//Alarm Word 24
(* uncomment when instrument is ready
Alarms_DB.AlarmWord_24.AlarmWord.0 := Trips_DB.Coil[9].ChargeRelay_FailtoClose; 
Alarms_DB.AlarmWord_24.AlarmWord.1 := Trips_DB.Coil[9].ChargeRelay_FailtoOpen;
Alarms_DB.AlarmWord_24.AlarmWord.2 := Trips_DB.Coil[10].ChargeRelay_FailtoClose;
Alarms_DB.AlarmWord_24.AlarmWord.3 := Trips_DB.Coil[10].ChargeRelay_FailtoOpen;
Alarms_DB.AlarmWord_24.AlarmWord.4 := Trips_DB.Coil[1].ACInterlockRelayFailedtoClose;
Alarms_DB.AlarmWord_24.AlarmWord.5 := Trips_DB.Coil[1].ACInterlockRelayFailedtoOpen;
Alarms_DB.AlarmWord_24.AlarmWord.6 := Trips_DB.Coil[2].ACInterlockRelayFailedtoClose;
Alarms_DB.AlarmWord_24.AlarmWord.7 := Trips_DB.Coil[2].ACInterlockRelayFailedtoOpen;
Alarms_DB.AlarmWord_24.AlarmWord.8 := Trips_DB.Coil[3].ACInterlockRelayFailedtoClose;
Alarms_DB.AlarmWord_24.AlarmWord.9 := Trips_DB.Coil[3].ACInterlockRelayFailedtoOpen;
Alarms_DB.AlarmWord_24.AlarmWord.10 := Trips_DB.Coil[4].ACInterlockRelayFailedtoClose;
Alarms_DB.AlarmWord_24.AlarmWord.11 := Trips_DB.Coil[4].ACInterlockRelayFailedtoOpen;
Alarms_DB.AlarmWord_24.AlarmWord.12 := Trips_DB.Coil[5].ACInterlockRelayFailedtoClose;
Alarms_DB.AlarmWord_24.AlarmWord.13 := Trips_DB.Coil[5].ACInterlockRelayFailedtoOpen;
Alarms_DB.AlarmWord_24.AlarmWord.14 := Trips_DB.Coil[6].ACInterlockRelayFailedtoClose;
Alarms_DB.AlarmWord_24.AlarmWord.15 := Trips_DB.Coil[6].ACInterlockRelayFailedtoOpen;
*)
//Alarm Word 24 msg
alarms[368](evtEntry:= Tc_Events.AlarmWord24.b0, bEvt:= Alarms_DB.AlarmWord_24.AlarmWord.0, bConfirm:= bConfirm);
alarms[369](evtEntry:= Tc_Events.AlarmWord24.b1, bEvt:= Alarms_DB.AlarmWord_24.AlarmWord.1, bConfirm:= bConfirm);
alarms[370](evtEntry:= Tc_Events.AlarmWord24.b2, bEvt:= Alarms_DB.AlarmWord_24.AlarmWord.2, bConfirm:= bConfirm);
alarms[371](evtEntry:= Tc_Events.AlarmWord24.b3, bEvt:= Alarms_DB.AlarmWord_24.AlarmWord.3, bConfirm:= bConfirm);
alarms[372](evtEntry:= Tc_Events.AlarmWord24.b4, bEvt:= Alarms_DB.AlarmWord_24.AlarmWord.4, bConfirm:= bConfirm);
alarms[373](evtEntry:= Tc_Events.AlarmWord24.b5, bEvt:= Alarms_DB.AlarmWord_24.AlarmWord.5, bConfirm:= bConfirm);
alarms[374](evtEntry:= Tc_Events.AlarmWord24.b6, bEvt:= Alarms_DB.AlarmWord_24.AlarmWord.6, bConfirm:= bConfirm);
alarms[375](evtEntry:= Tc_Events.AlarmWord24.b7, bEvt:= Alarms_DB.AlarmWord_24.AlarmWord.7, bConfirm:= bConfirm);
alarms[376](evtEntry:= Tc_Events.AlarmWord24.b8, bEvt:= Alarms_DB.AlarmWord_24.AlarmWord.8, bConfirm:= bConfirm);
alarms[377](evtEntry:= Tc_Events.AlarmWord24.b9, bEvt:= Alarms_DB.AlarmWord_24.AlarmWord.9, bConfirm:= bConfirm);
alarms[378](evtEntry:= Tc_Events.AlarmWord24.b10, bEvt:= Alarms_DB.AlarmWord_24.AlarmWord.10, bConfirm:= bConfirm);
alarms[379](evtEntry:= Tc_Events.AlarmWord24.b11, bEvt:= Alarms_DB.AlarmWord_24.AlarmWord.11, bConfirm:= bConfirm);
alarms[380](evtEntry:= Tc_Events.AlarmWord24.b12, bEvt:= Alarms_DB.AlarmWord_24.AlarmWord.12, bConfirm:= bConfirm);
alarms[381](evtEntry:= Tc_Events.AlarmWord24.b13, bEvt:= Alarms_DB.AlarmWord_24.AlarmWord.13, bConfirm:= bConfirm);
alarms[382](evtEntry:= Tc_Events.AlarmWord24.b14, bEvt:= Alarms_DB.AlarmWord_24.AlarmWord.14, bConfirm:= bConfirm);
alarms[383](evtEntry:= Tc_Events.AlarmWord24.b15, bEvt:= Alarms_DB.AlarmWord_24.AlarmWord.15, bConfirm:= bConfirm);

//Alarm Word 25
(* uncomment when instrument is ready
Alarms_DB.AlarmWord_25.AlarmWord.0 := Trips_DB.Coil[7].ACInterlockRelayFailedtoClose;
Alarms_DB.AlarmWord_25.AlarmWord.1 := Trips_DB.Coil[7].ACInterlockRelayFailedtoOpen;
Alarms_DB.AlarmWord_25.AlarmWord.2 := Trips_DB.Coil[8].ACInterlockRelayFailedtoClose;
Alarms_DB.AlarmWord_25.AlarmWord.3 := Trips_DB.Coil[8].ACInterlockRelayFailedtoOpen;
Alarms_DB.AlarmWord_25.AlarmWord.4 := Trips_DB.Coil[9].ACInterlockRelayFailedtoClose;
Alarms_DB.AlarmWord_25.AlarmWord.5 := Trips_DB.Coil[9].ACInterlockRelayFailedtoOpen;
Alarms_DB.AlarmWord_25.AlarmWord.6 := Trips_DB.Coil[10].ACInterlockRelayFailedtoClose;
Alarms_DB.AlarmWord_25.AlarmWord.7 := Trips_DB.Coil[10].ACInterlockRelayFailedtoOpen;
Alarms_DB.AlarmWord_25.AlarmWord.8 := Trips_DB.Coil[1].DumpRelay1_FailtoClose;
Alarms_DB.AlarmWord_25.AlarmWord.9 := Trips_DB.Coil[1].DumpRelay1_FailtoOpen;
Alarms_DB.AlarmWord_25.AlarmWord.10 := Trips_DB.Coil[2].DumpRelay1_FailtoClose;
Alarms_DB.AlarmWord_25.AlarmWord.11 := Trips_DB.Coil[2].DumpRelay1_FailtoOpen;
Alarms_DB.AlarmWord_25.AlarmWord.12 := Trips_DB.Coil[3].DumpRelay1_FailtoClose;
Alarms_DB.AlarmWord_25.AlarmWord.13 := Trips_DB.Coil[3].DumpRelay1_FailtoOpen;
Alarms_DB.AlarmWord_25.AlarmWord.14 := Trips_DB.Coil[4].DumpRelay1_FailtoClose;
Alarms_DB.AlarmWord_25.AlarmWord.15 := Trips_DB.Coil[4].DumpRelay1_FailtoOpen;
*)
//Alarm Word 25 msg
alarms[384](evtEntry:= Tc_Events.AlarmWord25.b0, bEvt:= Alarms_DB.AlarmWord_25.AlarmWord.0, bConfirm:= bConfirm);
alarms[385](evtEntry:= Tc_Events.AlarmWord25.b1, bEvt:= Alarms_DB.AlarmWord_25.AlarmWord.1, bConfirm:= bConfirm);
alarms[386](evtEntry:= Tc_Events.AlarmWord25.b2, bEvt:= Alarms_DB.AlarmWord_25.AlarmWord.2, bConfirm:= bConfirm);
alarms[387](evtEntry:= Tc_Events.AlarmWord25.b3, bEvt:= Alarms_DB.AlarmWord_25.AlarmWord.3, bConfirm:= bConfirm);
alarms[388](evtEntry:= Tc_Events.AlarmWord25.b4, bEvt:= Alarms_DB.AlarmWord_25.AlarmWord.4, bConfirm:= bConfirm);
alarms[389](evtEntry:= Tc_Events.AlarmWord25.b5, bEvt:= Alarms_DB.AlarmWord_25.AlarmWord.5, bConfirm:= bConfirm);
alarms[390](evtEntry:= Tc_Events.AlarmWord25.b6, bEvt:= Alarms_DB.AlarmWord_25.AlarmWord.6, bConfirm:= bConfirm);
alarms[391](evtEntry:= Tc_Events.AlarmWord25.b7, bEvt:= Alarms_DB.AlarmWord_25.AlarmWord.7, bConfirm:= bConfirm);
alarms[392](evtEntry:= Tc_Events.AlarmWord25.b8, bEvt:= Alarms_DB.AlarmWord_25.AlarmWord.8, bConfirm:= bConfirm);
alarms[393](evtEntry:= Tc_Events.AlarmWord25.b9, bEvt:= Alarms_DB.AlarmWord_25.AlarmWord.9, bConfirm:= bConfirm);
alarms[394](evtEntry:= Tc_Events.AlarmWord25.b10, bEvt:= Alarms_DB.AlarmWord_25.AlarmWord.10, bConfirm:= bConfirm);
alarms[395](evtEntry:= Tc_Events.AlarmWord25.b11, bEvt:= Alarms_DB.AlarmWord_25.AlarmWord.11, bConfirm:= bConfirm);
alarms[396](evtEntry:= Tc_Events.AlarmWord25.b12, bEvt:= Alarms_DB.AlarmWord_25.AlarmWord.12, bConfirm:= bConfirm);
alarms[397](evtEntry:= Tc_Events.AlarmWord25.b13, bEvt:= Alarms_DB.AlarmWord_25.AlarmWord.13, bConfirm:= bConfirm);
alarms[398](evtEntry:= Tc_Events.AlarmWord25.b14, bEvt:= Alarms_DB.AlarmWord_25.AlarmWord.14, bConfirm:= bConfirm);
alarms[399](evtEntry:= Tc_Events.AlarmWord25.b15, bEvt:= Alarms_DB.AlarmWord_25.AlarmWord.15, bConfirm:= bConfirm);

//Alarm Word 26
(* uncomment when instrument is ready
Alarms_DB.AlarmWord_26.AlarmWord.0 := Trips_DB.Coil[5].DumpRelay1_FailtoClose;
Alarms_DB.AlarmWord_26.AlarmWord.1 := Trips_DB.Coil[5].DumpRelay1_FailtoOpen;
Alarms_DB.AlarmWord_26.AlarmWord.2 := Trips_DB.Coil[6].DumpRelay1_FailtoClose;
Alarms_DB.AlarmWord_26.AlarmWord.3 := Trips_DB.Coil[6].DumpRelay1_FailtoOpen;
Alarms_DB.AlarmWord_26.AlarmWord.4 := Trips_DB.Coil[7].DumpRelay1_FailtoClose;
Alarms_DB.AlarmWord_26.AlarmWord.5 := Trips_DB.Coil[7].DumpRelay1_FailtoOpen;
Alarms_DB.AlarmWord_26.AlarmWord.6 := Trips_DB.Coil[8].DumpRelay1_FailtoClose;
Alarms_DB.AlarmWord_26.AlarmWord.7 := Trips_DB.Coil[8].DumpRelay1_FailtoOpen;
Alarms_DB.AlarmWord_26.AlarmWord.8 := Trips_DB.Coil[9].DumpRelay1_FailtoClose;
Alarms_DB.AlarmWord_26.AlarmWord.9 := Trips_DB.Coil[9].DumpRelay1_FailtoOpen;
Alarms_DB.AlarmWord_26.AlarmWord.10 := Trips_DB.Coil[10].DumpRelay1_FailtoClose;
Alarms_DB.AlarmWord_26.AlarmWord.11 := Trips_DB.Coil[10].DumpRelay1_FailtoOpen;
Alarms_DB.AlarmWord_26.AlarmWord.12 := Trips_DB.Coil[1].DumpRelay2_FailtoClose;
Alarms_DB.AlarmWord_26.AlarmWord.13 := Trips_DB.Coil[1].DumpRelay2_FailtoOpen;
Alarms_DB.AlarmWord_26.AlarmWord.14 := Trips_DB.Coil[2].DumpRelay2_FailtoClose;
Alarms_DB.AlarmWord_26.AlarmWord.15 := Trips_DB.Coil[2].DumpRelay2_FailtoOpen;
*)
//Alarm Word 26 msg
alarms[400](evtEntry:= Tc_Events.AlarmWord26.b0, bEvt:= Alarms_DB.AlarmWord_26.AlarmWord.0, bConfirm:= bConfirm);
alarms[401](evtEntry:= Tc_Events.AlarmWord26.b1, bEvt:= Alarms_DB.AlarmWord_26.AlarmWord.1, bConfirm:= bConfirm);
alarms[402](evtEntry:= Tc_Events.AlarmWord26.b2, bEvt:= Alarms_DB.AlarmWord_26.AlarmWord.2, bConfirm:= bConfirm);
alarms[403](evtEntry:= Tc_Events.AlarmWord26.b3, bEvt:= Alarms_DB.AlarmWord_26.AlarmWord.3, bConfirm:= bConfirm);
alarms[404](evtEntry:= Tc_Events.AlarmWord26.b4, bEvt:= Alarms_DB.AlarmWord_26.AlarmWord.4, bConfirm:= bConfirm);
alarms[405](evtEntry:= Tc_Events.AlarmWord26.b5, bEvt:= Alarms_DB.AlarmWord_26.AlarmWord.5, bConfirm:= bConfirm);
alarms[406](evtEntry:= Tc_Events.AlarmWord26.b6, bEvt:= Alarms_DB.AlarmWord_26.AlarmWord.6, bConfirm:= bConfirm);
alarms[407](evtEntry:= Tc_Events.AlarmWord26.b7, bEvt:= Alarms_DB.AlarmWord_26.AlarmWord.7, bConfirm:= bConfirm);
alarms[408](evtEntry:= Tc_Events.AlarmWord26.b8, bEvt:= Alarms_DB.AlarmWord_26.AlarmWord.8, bConfirm:= bConfirm);
alarms[409](evtEntry:= Tc_Events.AlarmWord26.b9, bEvt:= Alarms_DB.AlarmWord_26.AlarmWord.9, bConfirm:= bConfirm);
alarms[410](evtEntry:= Tc_Events.AlarmWord26.b10, bEvt:= Alarms_DB.AlarmWord_26.AlarmWord.10, bConfirm:= bConfirm);
alarms[411](evtEntry:= Tc_Events.AlarmWord26.b11, bEvt:= Alarms_DB.AlarmWord_26.AlarmWord.11, bConfirm:= bConfirm);
alarms[412](evtEntry:= Tc_Events.AlarmWord26.b12, bEvt:= Alarms_DB.AlarmWord_26.AlarmWord.12, bConfirm:= bConfirm);
alarms[413](evtEntry:= Tc_Events.AlarmWord26.b13, bEvt:= Alarms_DB.AlarmWord_26.AlarmWord.13, bConfirm:= bConfirm);
alarms[414](evtEntry:= Tc_Events.AlarmWord26.b14, bEvt:= Alarms_DB.AlarmWord_26.AlarmWord.14, bConfirm:= bConfirm);
alarms[415](evtEntry:= Tc_Events.AlarmWord26.b15, bEvt:= Alarms_DB.AlarmWord_26.AlarmWord.15, bConfirm:= bConfirm);

//Alarm Word 27
(* uncomment when instrument is ready
Alarms_DB.AlarmWord_27.AlarmWord.0 := Trips_DB.Coil[3].DumpRelay2_FailtoClose;
Alarms_DB.AlarmWord_27.AlarmWord.1 := Trips_DB.Coil[3].DumpRelay2_FailtoOpen;
Alarms_DB.AlarmWord_27.AlarmWord.2 := Trips_DB.Coil[4].DumpRelay2_FailtoClose;
Alarms_DB.AlarmWord_27.AlarmWord.3 := Trips_DB.Coil[4].DumpRelay2_FailtoOpen;
Alarms_DB.AlarmWord_27.AlarmWord.4 := Trips_DB.Coil[5].DumpRelay2_FailtoClose;
Alarms_DB.AlarmWord_27.AlarmWord.5 := Trips_DB.Coil[5].DumpRelay2_FailtoOpen;
Alarms_DB.AlarmWord_27.AlarmWord.6 := Trips_DB.Coil[6].DumpRelay2_FailtoClose;
Alarms_DB.AlarmWord_27.AlarmWord.7 := Trips_DB.Coil[6].DumpRelay2_FailtoOpen;
Alarms_DB.AlarmWord_27.AlarmWord.8 := Trips_DB.Coil[7].DumpRelay2_FailtoClose;
Alarms_DB.AlarmWord_27.AlarmWord.9 := Trips_DB.Coil[7].DumpRelay2_FailtoOpen;
Alarms_DB.AlarmWord_27.AlarmWord.10 := Trips_DB.Coil[8].DumpRelay2_FailtoClose;
Alarms_DB.AlarmWord_27.AlarmWord.11 := Trips_DB.Coil[8].DumpRelay2_FailtoOpen;
Alarms_DB.AlarmWord_27.AlarmWord.12:= Trips_DB.Coil[9].DumpRelay2_FailtoClose;
Alarms_DB.AlarmWord_27.AlarmWord.13 := Trips_DB.Coil[9].DumpRelay2_FailtoOpen;
Alarms_DB.AlarmWord_27.AlarmWord.14 := Trips_DB.Coil[10].DumpRelay2_FailtoClose;
Alarms_DB.AlarmWord_27.AlarmWord.15 := Trips_DB.Coil[10].DumpRelay2_FailtoOpen;
*)
//Alarm Word 27 msg
alarms[416](evtEntry:= Tc_Events.AlarmWord27.b0, bEvt:= Alarms_DB.AlarmWord_27.AlarmWord.0, bConfirm:= bConfirm);
alarms[417](evtEntry:= Tc_Events.AlarmWord27.b1, bEvt:= Alarms_DB.AlarmWord_27.AlarmWord.1, bConfirm:= bConfirm);
alarms[418](evtEntry:= Tc_Events.AlarmWord27.b2, bEvt:= Alarms_DB.AlarmWord_27.AlarmWord.2, bConfirm:= bConfirm);
alarms[419](evtEntry:= Tc_Events.AlarmWord27.b3, bEvt:= Alarms_DB.AlarmWord_27.AlarmWord.3, bConfirm:= bConfirm);
alarms[420](evtEntry:= Tc_Events.AlarmWord27.b4, bEvt:= Alarms_DB.AlarmWord_27.AlarmWord.4, bConfirm:= bConfirm);
alarms[421](evtEntry:= Tc_Events.AlarmWord27.b5, bEvt:= Alarms_DB.AlarmWord_27.AlarmWord.5, bConfirm:= bConfirm);
alarms[422](evtEntry:= Tc_Events.AlarmWord27.b6, bEvt:= Alarms_DB.AlarmWord_27.AlarmWord.6, bConfirm:= bConfirm);
alarms[423](evtEntry:= Tc_Events.AlarmWord27.b7, bEvt:= Alarms_DB.AlarmWord_27.AlarmWord.7, bConfirm:= bConfirm);
alarms[424](evtEntry:= Tc_Events.AlarmWord27.b8, bEvt:= Alarms_DB.AlarmWord_27.AlarmWord.8, bConfirm:= bConfirm);
alarms[425](evtEntry:= Tc_Events.AlarmWord27.b9, bEvt:= Alarms_DB.AlarmWord_27.AlarmWord.9, bConfirm:= bConfirm);
alarms[426](evtEntry:= Tc_Events.AlarmWord27.b10, bEvt:= Alarms_DB.AlarmWord_27.AlarmWord.10, bConfirm:= bConfirm);
alarms[427](evtEntry:= Tc_Events.AlarmWord27.b11, bEvt:= Alarms_DB.AlarmWord_27.AlarmWord.11, bConfirm:= bConfirm);
alarms[428](evtEntry:= Tc_Events.AlarmWord27.b12, bEvt:= Alarms_DB.AlarmWord_27.AlarmWord.12, bConfirm:= bConfirm);
alarms[429](evtEntry:= Tc_Events.AlarmWord27.b13, bEvt:= Alarms_DB.AlarmWord_27.AlarmWord.13, bConfirm:= bConfirm);
alarms[430](evtEntry:= Tc_Events.AlarmWord27.b14, bEvt:= Alarms_DB.AlarmWord_27.AlarmWord.14, bConfirm:= bConfirm);
alarms[431](evtEntry:= Tc_Events.AlarmWord27.b15, bEvt:= Alarms_DB.AlarmWord_27.AlarmWord.15, bConfirm:= bConfirm);
*)

//test
IF GVL.alarm_test THEN
	//i := i+1;
	Alarms_DB.MCP.AlarmWord := 16#FFFF;
	Alarms_DB.Section1.AlarmWord := 16#FFFF;
	Alarms_DB.Section2.AlarmWord := 16#FFFF;
	Alarms_DB.Section3.AlarmWord := 16#FFFF;
	Alarms_DB.Section4.AlarmWord := 16#FFFF;
	//Alarms_DB.Coil3.AlarmWord := 16#FFFF;
	//Alarms_DB.Coil4.AlarmWord := 16#FFFF;
	//Alarms_DB.Coil5.AlarmWord := 16#FFFF;
	//Alarms_DB.Coil6.AlarmWord := 16#FFFF;
	//Alarms_DB.Coil7.AlarmWord := 16#FFFF;
	//Alarms_DB.Coil8.AlarmWord := 16#FFFF;
	//Alarms_DB.Coil9.AlarmWord := 16#FFFF;
	//Alarms_DB.Coil10.AlarmWord := 16#FFFF;
	//Alarms_DB.AlarmWord_11.AlarmWord := 16#FFFF;
	//Alarms_DB.AlarmWord_22.AlarmWord := 16#FFFF;
	//Alarms_DB.AlarmWord_23.AlarmWord := 16#FFFF;
	//Alarms_DB.AlarmWord_24.AlarmWord := 16#FFFF;
	//Alarms_DB.AlarmWord_25.AlarmWord := 16#FFFF;
	//Alarms_DB.AlarmWord_26.AlarmWord := 16#FFFF;
	//Alarms_DB.AlarmWord_27.AlarmWord := 16#FFFF;
END_IF


//Clear Alarm Word
IF bConfirm THEN
	Alarms_DB.MCP.AlarmWord := 0;
	Alarms_DB.Section1.AlarmWord := 0;
	Alarms_DB.Section2.AlarmWord := 0;
	Alarms_DB.Section3.AlarmWord := 0;
	Alarms_DB.Section4.AlarmWord := 0;
	(*Alarms_DB.Coil3.AlarmWord := 0;
	Alarms_DB.Coil4.AlarmWord := 0;
	Alarms_DB.Coil5.AlarmWord := 0;
	Alarms_DB.Coil6.AlarmWord := 0;
	Alarms_DB.Coil7.AlarmWord := 0;
	Alarms_DB.Coil8.AlarmWord := 0;
	Alarms_DB.Coil9.AlarmWord := 0;
	Alarms_DB.Coil10.AlarmWord := 0;
	Alarms_DB.AlarmWord_11.AlarmWord := 0;
	Alarms_DB.AlarmWord_22.AlarmWord := 0;
	Alarms_DB.AlarmWord_23.AlarmWord := 0;
	Alarms_DB.AlarmWord_24.AlarmWord := 0;
	Alarms_DB.AlarmWord_25.AlarmWord := 0;
	Alarms_DB.AlarmWord_26.AlarmWord := 0;
	Alarms_DB.AlarmWord_27.AlarmWord := 0;
	*)
END_IF;

END_PROGRAM

// ---- POUs/Sequence.TcPOU
PROGRAM Sequence
VAR
	ePulseState : E_PulseState;
	//eCommand	: E_Command;
	i : INT := 1; //1-8 chargers
	j : INT := 1; //section 1-3
	k : INT := 1; //section 1- 4 
	
	//ChrgRlyHVON_TON : TON;
	//ChrgRlyHVON_PT 	: TIME := T#250MS;
	//ChrgRlyHVON_ET 	: TIME;
END_VAR


//charge command from screen room
IF MCP_IO.CloseAllChargeRlyCommand = TRUE THEN
	//CLOSE ALL CHARGE RELAYS	
	FOR j := 1 TO 3 BY 1 DO
		LCP.Section[j].Peak.CloseChargeRelay1 := TRUE;
		LCP.Section[j].Peak.CloseChargeRelay2 := TRUE;
		LCP.Section[j].Sust.CloseChargeRelay1 := TRUE;
		LCP.Section[j].Sust.CloseChargeRelay2 := TRUE;
	END_FOR;
	LCP.Section[4].Form.CloseChargeRelay1 := TRUE;
	LCP.Section[4].Form.CloseChargeRelay2 := TRUE;
							
	LCP.Section[4].Form.ClosePreFormChargeRly := TRUE;
	LCP.Section[4].Form.CloseFormTrigChargeRly := TRUE;
	LCP.Section[4].Form.ClosePreFormTrigChargeRly := TRUE;
				
ELSE
	//OPEN ALL CHARGE RELAYS	
	FOR j := 1 TO 3 BY 1 DO
		LCP.Section[j].Peak.CloseChargeRelay1 := FALSE;
		LCP.Section[j].Peak.CloseChargeRelay2 := FALSE;
		LCP.Section[j].Sust.CloseChargeRelay1 := FALSE;
		LCP.Section[j].Sust.CloseChargeRelay2 := FALSE;
	END_FOR;
	LCP.Section[4].Form.CloseChargeRelay1 := FALSE;
	LCP.Section[4].Form.CloseChargeRelay2 := FALSE;
							
	LCP.Section[4].Form.ClosePreFormChargeRly := FALSE;
	LCP.Section[4].Form.CloseFormTrigChargeRly := FALSE;
	LCP.Section[4].Form.ClosePreFormTrigChargeRly := FALSE;
END_IF;

//use this for the slim only  -- it will be replaced with the Permissives block for the next upgrade
(*IF Permissives_DB.AllChargeRelaysClosed = TRUE THEN 
		//system ready to charge LED On
		FOR k := 1 TO 4	BY 1 DO 
			LCP.Section[k].SystemReadyToCharge := TRUE;
		END_FOR;
	ELSE
		//system ready to charge LED On
		FOR k := 1 TO 4	BY 1 DO 
			LCP.Section[k].SystemReadyToCharge := FALSE;
		END_FOR;
END_IF;
*)
//open dump command from screen room
IF MCP_IO.OpenAllDumpRelayCommand = TRUE THEN			
	//Open all dump relays 
	FOR j := 1 TO 3 BY 1 DO						
		LCP.Section[j].Peak.OpenDumpRelay1 := TRUE;
		LCP.Section[j].Peak.OpenDumpRelay2 := TRUE;
		LCP.Section[j].Sust.OpenDumpRelay1 := TRUE;
		LCP.Section[j].Sust.OpenDumpRelay2 := TRUE;
							
		LCP.Section[4].Form.OpenDumpRelay1 := TRUE;
		LCP.Section[4].Form.OpenDumpRelay2 := TRUE;
		LCP.Section[4].Form.OpenPreFormDumpRly	:= TRUE;
		LCP.Section[4].Form.OpenFormTrigDumpRly1 := TRUE;
		LCP.Section[4].Form.OpenPreFormTrigDumpRly1 := TRUE;
	END_FOR;
ELSE
	//Close all dump relays 
	FOR j := 1 TO 3 BY 1 DO						
		LCP.Section[j].Peak.OpenDumpRelay1 := FALSE;
		LCP.Section[j].Peak.OpenDumpRelay2 := FALSE;
		LCP.Section[j].Sust.OpenDumpRelay1 := FALSE;
		LCP.Section[j].Sust.OpenDumpRelay2 := FALSE;
							
		LCP.Section[4].Form.OpenDumpRelay1 := FALSE;
		LCP.Section[4].Form.OpenDumpRelay2 := FALSE;
		LCP.Section[4].Form.OpenPreFormDumpRly	:= FALSE;
		LCP.Section[4].Form.OpenFormTrigDumpRly1 := FALSE;
		LCP.Section[4].Form.OpenPreFormTrigDumpRly1 := FALSE;
	END_FOR;
END_IF;

//mapping to the MCP for slim configuration
MCP_IO.AllChargeRelaysClose := Permissives_DB.AllChargeRelaysClosed;
MCP_IO.AllDumpRelaysOpen := Permissives_DB.AllDumpRelaysOpen;


//no sequencing needed************************************************************************************************
(*
//IF BOTH Close charge and open dump signals are off go to idle.
IF MCP_IO.CloseAllChargeRlyCommand = FALSE AND MCP_IO.OpenAllDumpRelayCommand = FALSE THEN
	ePulseState := E_PulseState.SAFE;
END_IF;




//screen room asks to go to close all charge relays when the dump relays are closed ** this should never happen
IF MCP_IO.CloseAllChargeRlyCommand = TRUE AND MCP_IO.OpenAllDumpRelayCommand = FALSE THEN
	ePulseState := E_PulseState.TRIPPED;
END_IF;

//screen room asks to go to open all charge relays when the dump relays are open ** this should never happen - floating system
(*
IF MCP_IO.CloseAllChargeRlyCommand = FALSE AND MCP_IO.OpenAllDumpRelayCommand = TRUE THEN
	//both charge and dump open - floating
END_IF;
*)


CASE ePulseState OF 
	//SAFE / IDLE state
	E_PulseState.SAFE:
							
						//IF no fault and charge permissions and charge relay go to charge mode
						IF MCP_IO.CloseAllChargeRlyCommand = TRUE AND MCP_IO.OpenAllDumpRelayCommand = TRUE THEN
							ePulseState := E_PulseState.CHARGING;
						END_IF;

	//CHARGING STATE
	E_PulseState.CHARGING:
							//turn on charger inhibit
							FOR i := 1 TO 8 BY 1 DO
								MCP_IO.Charger[i].inhibit := TRUE;
							END_FOR;
							
							//Open all dump relays first
							LCP.Bank[j].Peak.OpenDumpRelay1 := TRUE;
							LCP.Bank[j].Peak.OpenDumpRelay2 := TRUE;
							LCP.Bank[j].Sust.OpenDumpRelay1 := TRUE;
							LCP.Bank[j].Sust.OpenDumpRelay2 := TRUE;
							
							LCP.Bank[4].Form.OpenDumpRelay1 := TRUE;
							LCP.Bank[4].Form.OpenDumpRelay2 := TRUE;
							LCP.Bank[4].OpenPreFormDumpRly	:= TRUE;
							LCP.Bank[4].OpenFormTrigDumpRly1 := TRUE;
							LCP.Bank[4].OpenPreFormTrigDumpRly1 := TRUE;
							
							
							
							
							
							//CLOSE ALL CHARGE RELAYS	
							FOR j := 1 TO 3 BY 1 DO
								LCP.Bank[j].Peak.CloseChargeRelay1 := TRUE;
								LCP.Bank[j].Peak.CloseChargeRelay2 := TRUE;
								LCP.Bank[j].Sust.CloseChargeRelay1 := TRUE;
								LCP.Bank[j].Sust.CloseChargeRelay2 := TRUE;
							END_FOR;
							LCP.Bank[4].Form.CloseChargeRelay1 := TRUE;
							LCP.Bank[4].Form.CloseChargeRelay2 := TRUE;
							
							LCP.Bank[4].ClosePreFormChargeRly := TRUE;
							LCP.Bank[4].CloseFormTrigChargeRly := TRUE;
							LCP.Bank[4].ClosePreFormTrigChargeRly := TRUE;
				
							IF MCP_IO.AllChargeRelaysClose = TRUE THEN
								//system ready to charge LED On
								FOR k := 1 TO 4	BY 1 DO 
									LCP.Bank[k].SystemReadyToCharge := TRUE;
								END_FOR;							
						
								//enable all HV ON output and remove inhitbit signal
								FOR i := 1 TO 8 BY 1 DO 
									MCP_IO.Charger[i].HV_ON := TRUE;
									MCP_IO.Charger[i].inhibit := TRUE;
								END_FOR;
								
							ELSE 
								//system ready to charge LED Off
								FOR k := 1 TO 4	BY 1 DO 
									LCP.Bank[k].SystemReadyToCharge := FALSE;
								END_FOR;
									
								FOR i := 1 TO 8 BY 1 DO 
									MCP_IO.Charger[i].HV_ON := FALSE;
								END_FOR;
							END_IF;
							
							//if screen room ask to go the dump
							IF MCP_IO.OpenAllDumpRelayCommand = FALSE AND MCP_IO.CloseAllChargeRlyCommand = FALSE THEN
								ePulseState := E_PulseState.DUMPING;
							END_IF;
	
	//DUMP STATE
	E_PulseState.DUMPING:
							//turn off charger HV ON and Inhibit signals
							FOR i := 1 TO 8 BY 1 DO 
								MCP_IO.Charger[i].HV_ON := FALSE;
								MCP_IO.Charger[i].inhibit := FALSE;
							END_FOR; 
							
							IF MCP_IO.AllChargerHVisON = FALSE THEN
								//Open ALL CHARGE RELAYS	
								FOR j := 1 TO 3 BY 1 DO
									LCP.Bank[j].Peak.CloseChargeRelay1 := FALSE;
									LCP.Bank[j].Peak.CloseChargeRelay2 := FALSE;
									LCP.Bank[j].Sust.CloseChargeRelay1 := FALSE;
									LCP.Bank[j].Sust.CloseChargeRelay2 := FALSE;
								END_FOR;
								LCP.Bank[4].Form.CloseChargeRelay1 := FALSE;
								LCP.Bank[4].Form.CloseChargeRelay2 := FALSE;
							
								LCP.Bank[4].ClosePreFormChargeRly := FALSE;
								LCP.Bank[4].CloseFormTrigChargeRly := FALSE;
								LCP.Bank[4].ClosePreFormTrigChargeRly := FALSE;
							END_IF;
							
							FOR j := 1 TO 3 BY 1 DO 
								LCP.Bank[j].Peak.OpenDumpRelay1 := FALSE;
								LCP.Bank[j].Peak.OpenDumpRelay2 := TRUE;
								LCP.Bank[j].Peak.OpenDumpRelay2 := TRUE;
							END_FOR;
						
	
	//TRIPPED STATE
	E_PulseState.TRIPPED:
							//DO SOMETHING
	
	
	
	
	
END_CASE;
*)
//**********************************************************************************	




IF i > 8 THEN
	i := 1;
END_IF;

IF j > 3 THEN
	j := 1;
END_IF;

IF k > 4 THEN
	k := 1;
END_IF;

END_PROGRAM
